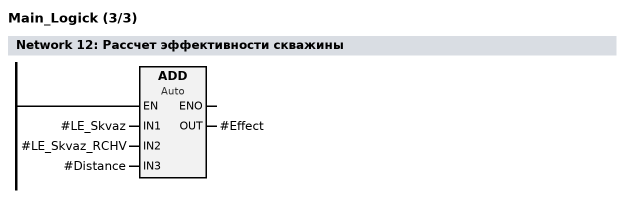
   RUNG wire#powerrail
      Add(in1 := #LE_Skvaz, in2 := #LE_Skvaz_RCHV, in3 := #Distance, out => #Effect)
   END_RUNG
   // the same network as SCL:
   #Effect := #LE_Skvaz + #LE_Skvaz_RCHV + #Distance;
END_REGION
END_FUNCTION_BLOCK

FUNCTION "Pump_LE" : Void
{ S7_Optimized_Access := 'TRUE' }
VERSION : 0.1
   VAR_INPUT 
      Level_Norm : Real;
      LS : Real;
      LE_now : Real;
   END_VAR

   VAR_TEMP 
      x : Array[1..10] of Real;
      Delta : Real;
   END_VAR


BEGIN
	//рассчёт коррекции при падении уровня в РЧВ
	#x[1] := #Level_Norm - #LS;
	#x[2] := #LE_now - #LS;
	#x[3] := #x[1] / #x[2];
	#Delta := 1 - #x[3];
	
	//уровень ниже рабочей точки
	IF #Delta < 1.0 THEN
	    "Main_Logick_DB".Alarms.LE_Warning := TRUE;
	ELSE
	    "Main_Logick_DB".Alarms.LE_Warning := FALSE;
	    #Delta := 1.0;
	END_IF;
	
	//уровень в аварийной зоне
	IF #Delta <= 0.0 THEN
	    "Main_Logick_DB".Alarms.LE_Alarm := TRUE;
	    #Delta := 0.0;
	ELSE
	    "Main_Logick_DB".Alarms.LE_Alarm := FALSE;
	END_IF;
	
	//коррекция уставки при аварийных ситуациях
	IF "Main_Logick_DB".Mode = TRUE THEN
	    "Pump_DB".SP_A := "Main_Logick_DB".PID_Pump.Result * #Delta;
	ELSE
	    "Pump_DB".SP_A := "Main_Logick_DB".SP_Pump * #Delta;
	END_IF;
END_FUNCTION

FUNCTION_BLOCK "DRV_Flow"   // FB130, LAD
{ S7_Optimized_Access := 'FALSE' }
VERSION : 0.1
// stored: AutoNumber false, IsIECCheckEnabled false, SetENOAutomatically false, UDAEnableTagReadback false
   VAR_IN_OUT
      impulse : Bool;
      FlowSpeed : Real;
   END_VAR
   VAR DB_SPECIFIC
      CMD : "CMD";
      Mode : Int;   // 0 - л/м, 1- л/ч, 2- м3/ч / Режим работы
      Status : Int;   // Статус устройства
      Use : Struct   // Функционал
         Indirect { S7_SetPoint := 'True'} : Bool := true;
         call_in_OB1 { S7_SetPoint := 'True'} : Bool := true;
      END_STRUCT;
      Clock { S7_SetPoint := 'True'} : Real := 0.1;   // Частота измерений
      Weight { S7_SetPoint := 'True'} : Real := 1.0;   // Вес импульса
      Time_Now : Real;
      Time_Last : Real;
      Time_Mid : Real;
      Flow_S : Real;   // литры в секунду
      Alarms : Word;   // Слово аварий
      Events : Word;   // События
      ADDR_BYTE { S7_SetPoint := 'True'} : Int;
      ADDR_BIT { S7_SetPoint := 'True'} : Int := 9;
   END_VAR
   VAR
      Filter { S7_SetPoint := 'True'} : "Filter";
   END_VAR
   VAR DB_SPECIFIC
      pos : Array[0..15] of Bool;
      "Name" { S7_SetPoint := 'True'} : String[4];
      Time_DTL : DTL;
   END_VAR
   VAR_TEMP
      imp : Bool;
      Filter_clock : Bool;
   END_VAR
   VAR CONSTANT
      sec : Int := 60;
   END_VAR
   // Filter.max := 100;
   VAR_TEMP   // added for the SCL form of the ladder/FBD networks
      _w1 : Bool;
      _w2 : Bool;
      _w3 : Bool;
   END_VAR
BEGIN

REGION Network 1: Чтение входа
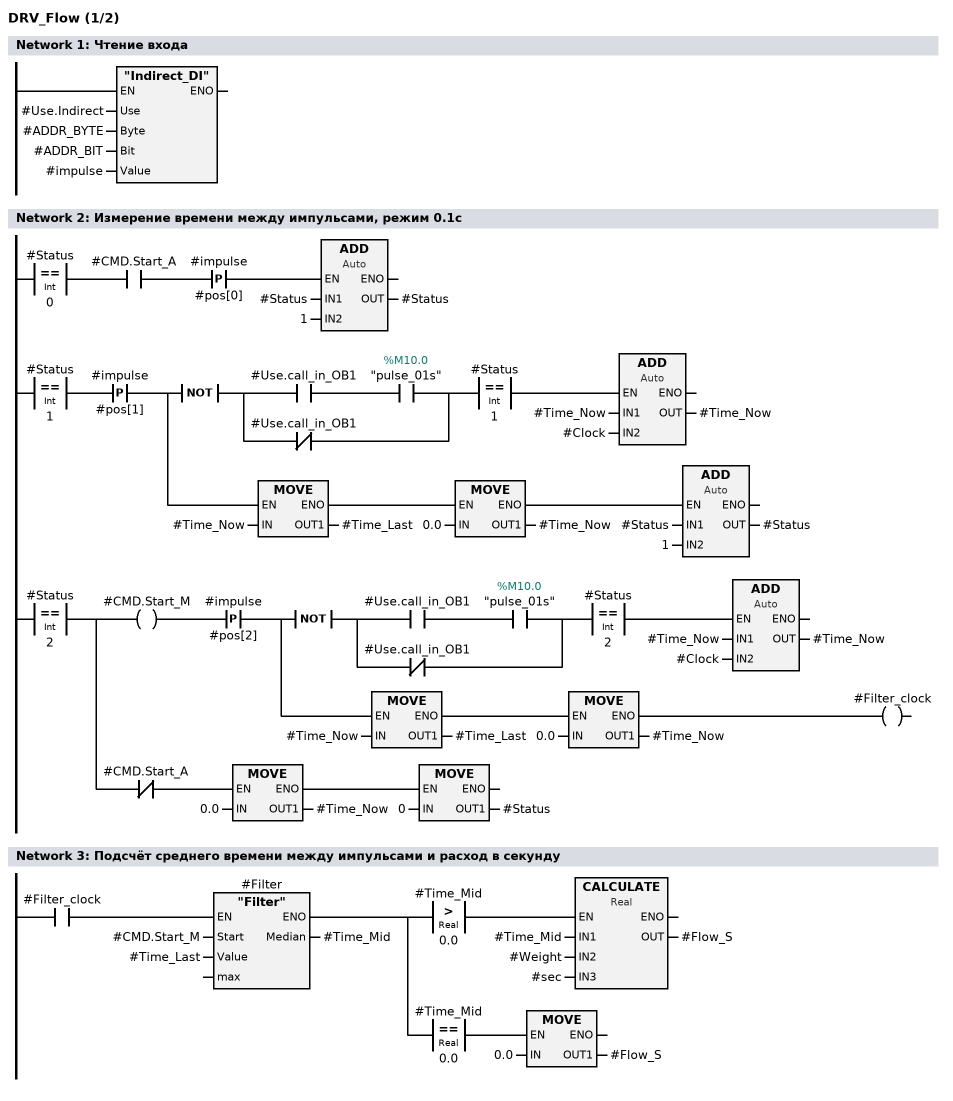
   RUNG wire#powerrail
      "Indirect_DI"(Use := #Use.Indirect, "Byte" := #ADDR_BYTE, Bit := #ADDR_BIT, Value := #impulse)
   END_RUNG
   // the same network as SCL:
   "Indirect_DI"(Use := #Use.Indirect, "Byte" := #ADDR_BYTE, Bit := #ADDR_BIT, Value := #impulse);
END_REGION

REGION Network 2: Измерение времени между импульсами, режим 0.1с
   RUNG wire#powerrail
      { S7_Templates := "SrcType := Int" } EQ_Contact(in1 := #Status, in2 := 0)
      Contact( #CMD.Start_A )
      P_Contact(operand := #impulse, bit := #pos[0])
      Add(in1 := #Status, in2 := 1, out => #Status)
   END_RUNG
   RUNG wire#powerrail
      { S7_Templates := "SrcType := Int" } EQ_Contact(in1 := #Status, in2 := 1)
      P_Contact(operand := #impulse, bit := #pos[1])
      wire#w1
      Not()
      wire#w2
      Contact( #Use.call_in_OB1 )
      Contact( "pulse_01s" )
      wire#w3
      { S7_Templates := "SrcType := Int" } EQ_Contact(in1 := #Status, in2 := 1)
      Add(in1 := #Time_Now, in2 := #Clock, out => #Time_Now)
   END_RUNG
   RUNG wire#w2
      I_Contact( #Use.call_in_OB1 )
   END_RUNG wire#w3
   RUNG wire#w1
      Move(in := #Time_Now, out1 => #Time_Last)
      Move(in := 0.0, out1 => #Time_Now)
      Add(in1 := #Status, in2 := 1, out => #Status)
   END_RUNG
   RUNG wire#powerrail
      { S7_Templates := "SrcType := Int" } EQ_Contact(in1 := #Status, in2 := 2)
      wire#w4
      Coil( #CMD.Start_M )
      P_Contact(operand := #impulse, bit := #pos[2])
      wire#w5
      Not()
      wire#w6
      Contact( #Use.call_in_OB1 )
      Contact( "pulse_01s" )
      wire#w7
      { S7_Templates := "SrcType := Int" } EQ_Contact(in1 := #Status, in2 := 2)
      Add(in1 := #Time_Now, in2 := #Clock, out => #Time_Now)
   END_RUNG
   RUNG wire#w6
      I_Contact( #Use.call_in_OB1 )
   END_RUNG wire#w7
   RUNG wire#w5
      Move(in := #Time_Now, out1 => #Time_Last)
      Move(in := 0.0, out1 => #Time_Now)
      Coil( #Filter_clock )
   END_RUNG
   RUNG wire#w4
      I_Contact( #CMD.Start_A )
      Move(in := 0.0, out1 => #Time_Now)
      Move(in := 0, out1 => #Status)
   END_RUNG
   // the same network as SCL:
   #_w1 := (#Status = 0) AND #CMD.Start_A AND #impulse AND NOT #pos[0];   // rising edge of #impulse
   #pos[0] := #impulse;
   IF #_w1 THEN #Status := #Status + 1; END_IF;
   #_w2 := (#Status = 1) AND #impulse AND NOT #pos[1];   // rising edge of #impulse
   #pos[1] := #impulse;
   IF NOT #_w2 AND ((#Use.call_in_OB1 AND "pulse_01s") OR NOT #Use.call_in_OB1) AND (#Status = 1) THEN
       #Time_Now := #Time_Now + #Clock;
   END_IF;
   IF #_w2 THEN
       #Time_Last := #Time_Now;
       #Time_Now := 0.0;
       #Status := #Status + 1;
   END_IF;
   #CMD.Start_M := #Status = 2;
   #_w3 := #CMD.Start_M AND #impulse AND NOT #pos[2];   // rising edge of #impulse
   #pos[2] := #impulse;
   IF NOT #_w3 AND ((#Use.call_in_OB1 AND "pulse_01s") OR NOT #Use.call_in_OB1) AND (#Status = 2) THEN
       #Time_Now := #Time_Now + #Clock;
   END_IF;
   IF #_w3 THEN
       #Time_Last := #Time_Now;
       #Time_Now := 0.0;
   END_IF;
   #Filter_clock := #_w3;
   IF #CMD.Start_M AND NOT #CMD.Start_A THEN
       #Time_Now := 0.0;
       #Status := 0;
   END_IF;
END_REGION

REGION Network 3: Подсчёт среднего времени между импульсами и расход в секунду
   RUNG wire#powerrail
      Contact( #Filter_clock )
      #Filter(Start := #CMD.Start_M, Value := #Time_Last, max :=, Median => #Time_Mid)
      wire#w1
      { S7_Templates := "SrcType := Real" } GT_Contact(in1 := #Time_Mid, in2 := 0.0)
      { S7_Templates := "SrcType := Real"; S7_Expression := "IN3/IN1*IN2" } Calculate(in1 := #Time_Mid, in2 := #Weight, in3 := #sec, out => #Flow_S)
   END_RUNG
   RUNG wire#w1
      { S7_Templates := "SrcType := Real" } EQ_Contact(in1 := #Time_Mid, in2 := 0.0)
      Move(in := 0.0, out1 => #Flow_S)
   END_RUNG
   // the same network as SCL:
   #Filter(EN := #Filter_clock, Start := #CMD.Start_M, Value := #Time_Last, Median => #Time_Mid, ENO => #_w1);   // "Filter"
   IF #_w1 AND (#Time_Mid > 0.0) THEN #Flow_S := #sec/#Time_Mid*#Weight; END_IF;
   IF #_w1 AND (#Time_Mid = 0.0) THEN #Flow_S := 0.0; END_IF;
END_REGION

REGION Network 4: Расход л/м, л/ч, м3/ч
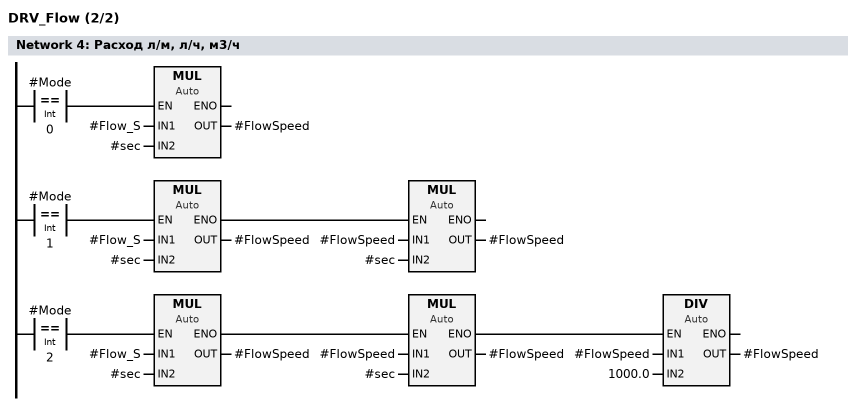
   RUNG wire#powerrail
      { S7_Templates := "SrcType := Int" } EQ_Contact(in1 := #Mode, in2 := 0)
      Mul(in1 := #Flow_S, in2 := #sec, out => #FlowSpeed)
   END_RUNG
   RUNG wire#powerrail
      { S7_Templates := "SrcType := Int" } EQ_Contact(in1 := #Mode, in2 := 1)
      Mul(in1 := #Flow_S, in2 := #sec, out => #FlowSpeed)
      Mul(in1 := #FlowSpeed, in2 := #sec, out => #FlowSpeed)
   END_RUNG
   RUNG wire#powerrail
      { S7_Templates := "SrcType := Int" } EQ_Contact(in1 := #Mode, in2 := 2)
      Mul(in1 := #Flow_S, in2 := #sec, out => #FlowSpeed)
      Mul(in1 := #FlowSpeed, in2 := #sec, out => #FlowSpeed)
      Div(in1 := #FlowSpeed, in2 := 1000.0, out => #FlowSpeed)
   END_RUNG
   // the same network as SCL:
   IF #Mode = 0 THEN #FlowSpeed := #Flow_S * #sec; END_IF;
   IF #Mode = 1 THEN
       #FlowSpeed := #Flow_S * #sec;
       #FlowSpeed := #FlowSpeed * #sec;
   END_IF;
   IF #Mode = 2 THEN
       #FlowSpeed := #Flow_S * #sec;
       #FlowSpeed := #FlowSpeed * #sec;
       #FlowSpeed := #FlowSpeed / 1000.0;
   END_IF;
END_REGION
END_FUNCTION_BLOCK

DATA_BLOCK "Comm_SKD1_DB"   // DB10
VERSION : 0.1
// stored: AutoNumber false, DBAccessibleFromOPCUA true, InstanceOfName Comm_SKD1, InstanceOfType FB
"Comm_SKD1"
BEGIN
   Valve_Name[1..10] := '';
END_DATA_BLOCK

DATA_BLOCK "Main_Logick_DB"   // DB1
VERSION : 0.1
// stored: AutoNumber true, DBAccessibleFromOPCUA true, InstanceOfName Main_Logick, InstanceOfType FB
"Main_Logick"
BEGIN
   PID_Pump.CMD.Vector := FALSE;
   PID_Pump.x := 1.0;
   PID_Pump.Settings.SP_P := 1.5;
   PID_Pump.Settings.SP_Ti := 150.0;
   PID_Pump.Settings.SP_Td := 0.0;
   PID_Pump.Settings.SP_Cycle := 0.2;
   PID_Pump.Settings.Max_SP := 500.0;
   PID_Pump.Settings.Min_SP := -500.0;
   PID_Pump.Settings.Max_in := 500.0;
   PID_Pump.Settings.Min_in := -500.0;
   PID_Pump.Settings.Max_out := 100.0;
   PID_Pump.Settings.Min_out := 0.0;
   PID_Pump.Settings.DeadBand := 1.0;
   PID_Pump.PID.IntegralResetMode := 4;
   PID_Pump.PID.RunModeByStartup := TRUE;
   PID_Pump.PID.SetSubstituteOutput := TRUE;
   PID_Pump.PID.ActivateRecoverMode := TRUE;
   PID_Pump.PID.CancelTuningLevel := 10.0;
   PID_Pump.PID.SubstituteOutput := 0.0;
   PID_Pump.PID.Config.InputPerOn := TRUE;
   PID_Pump.PID.Config.InvertControl := FALSE;
   PID_Pump.PID.Config.InputUpperLimit := 120.0;
   PID_Pump.PID.Config.InputLowerLimit := 0.0;
   PID_Pump.PID.Config.InputUpperWarning := 3.402822E+38;
   PID_Pump.PID.Config.InputLowerWarning := -3.402822E+38;
   PID_Pump.PID.Config.OutputUpperLimit := 100.0;
   PID_Pump.PID.Config.OutputLowerLimit := 0.0;
   PID_Pump.PID.Config.SetpointUpperLimit := 3.402822E+38;
   PID_Pump.PID.Config.SetpointLowerLimit := -3.402822E+38;
   PID_Pump.PID.Config.MinimumOnTime := 0.0;
   PID_Pump.PID.Config.MinimumOffTime := 0.0;
   PID_Pump.PID.Config.InputScaling.UpperPointIn := 27648.0;
   PID_Pump.PID.Config.InputScaling.LowerPointIn := 0.0;
   PID_Pump.PID.Config.InputScaling.UpperPointOut := 100.0;
   PID_Pump.PID.Config.InputScaling.LowerPointOut := 0.0;
   PID_Pump.PID.CycleTime.EnEstimation := TRUE;
   PID_Pump.PID.CycleTime.EnMonitoring := TRUE;
   PID_Pump.PID.CycleTime.Value := 0.1;
   PID_Pump.PID.CtrlParamsBackUp.Gain := 1.0;
   PID_Pump.PID.CtrlParamsBackUp.Ti := 20.0;
   PID_Pump.PID.CtrlParamsBackUp.Td := 0.0;
   PID_Pump.PID.CtrlParamsBackUp.TdFiltRatio := 0.2;
   PID_Pump.PID.CtrlParamsBackUp.PWeighting := 1.0;
   PID_Pump.PID.CtrlParamsBackUp.DWeighting := 1.0;
   PID_Pump.PID.CtrlParamsBackUp.Cycle := 1.0;
   PID_Pump.PID.PIDSelfTune.SUT.TuneRule := 0;
   PID_Pump.PID.PIDSelfTune.TIR.TuneRule := 0;
   PID_Pump.PID.Retain.CtrlParams.Gain := 1.0;
   PID_Pump.PID.Retain.CtrlParams.Ti := 20.0;
   PID_Pump.PID.Retain.CtrlParams.Td := 0.0;
   PID_Pump.PID.Retain.CtrlParams.TdFiltRatio := 0.2;
   PID_Pump.PID.Retain.CtrlParams.PWeighting := 1.0;
   PID_Pump.PID.Retain.CtrlParams.DWeighting := 1.0;
   PID_Pump.PID.Retain.CtrlParams.Cycle := 1.0;
   PID_Pump.C.SP := 1.0;
   PID_Pump.C.One := 0.1;
END_DATA_BLOCK

DATA_BLOCK "System_DB"   // DB4
VERSION : 0.1
// stored: AutoNumber true, DBAccessibleFromOPCUA true, InstanceOfName System, InstanceOfType FB
"System"
BEGIN
END_DATA_BLOCK

DATA_BLOCK "ModBus_DB"   // DB20
VERSION : 0.1
// stored: AutoNumber false, DBAccessibleFromOPCUA true, InstanceOfName ModBus, InstanceOfType FB
"ModBus"
BEGIN
END_DATA_BLOCK

DATA_BLOCK "ModBus_TCP_DB"   // DB40
VERSION : 0.1
// stored: AutoNumber false, DBAccessibleFromOPCUA true, InstanceOfName ModBus_TCP, InstanceOfType FB
"ModBus_TCP"
BEGIN
   DATA[0..100] := 16#0000;
   CONNECT.InterfaceId := 64;
   CONNECT.ID := 16#0001;
   CONNECT.ConnectionType := 16#0B;
   CONNECT.ActiveEstablished := TRUE;
   CONNECT.RemoteAddress.ADDR[1] := 16#0A;
   CONNECT.RemoteAddress.ADDR[2..3] := 16#01;
   CONNECT.RemoteAddress.ADDR[4] := 16#C9;
   CONNECT.RemotePort := 503;
   CONNECT.LocalPort := 0;
END_DATA_BLOCK

DATA_BLOCK "AIx_DB"   // DB220
VERSION : 0.1
// stored: AutoNumber false, DBAccessibleFromOPCUA true, InstanceOfName AIx, InstanceOfType FB
"AIx"
BEGIN
END_DATA_BLOCK

DATA_BLOCK "DIx_1_DB"   // DB200
VERSION : 0.1
// stored: AutoNumber false, DBAccessibleFromOPCUA true, InstanceOfName DIx_1, InstanceOfType FB
"DIx_1"
BEGIN
   AllBlock.Use.Inverse := FALSE;
   AllBlock.Use.Indirect := TRUE;
   AllBlock.ADDR_Byte := 0;
   AllBlock.ADDR_Bit := 3;
   AllBlock.Filter_On.SP := 16#02;
   AllBlock.Filter_Off.SP := 16#02;
   "3FOk".Use.Inverse := FALSE;
   "3FOk".Use.Indirect := TRUE;
   "3FOk".ADDR_Byte := 0;
   "3FOk".ADDR_Bit := 0;
   "3FOk".Filter_On.SP := 16#02;
   "3FOk".Filter_Off.SP := 16#02;
   Pump_Alarm.Use.Inverse := FALSE;
   Pump_Alarm.Use.Indirect := TRUE;
   Pump_Alarm.ADDR_Byte := 0;
   Pump_Alarm.ADDR_Bit := 2;
   Pump_Alarm.Filter_On.SP := 16#02;
   Pump_Alarm.Filter_Off.SP := 16#02;
   Leak_KP.Use.Inverse := FALSE;
   Leak_KP.Use.Indirect := TRUE;
   Leak_KP.ADDR_Byte := 0;
   Leak_KP.ADDR_Bit := 4;
   Leak_KP.Filter_On.SP := 16#02;
   Leak_KP.Filter_Off.SP := 16#02;
   Level_Norm.Use.Inverse := FALSE;
   Level_Norm.Use.Indirect := TRUE;
   Level_Norm.ADDR_Byte := 0;
   Level_Norm.ADDR_Bit := 5;
   Level_Norm.Filter_On.SP := 16#02;
   Level_Norm.Filter_Off.SP := 16#02;
   "3Fok_1".Use.Inverse := FALSE;
   "3Fok_1".Use.Indirect := TRUE;
   "3Fok_1".ADDR_Byte := 0;
   "3Fok_1".ADDR_Bit := 6;
   "3Fok_1".Filter_On.SP := 16#02;
   "3Fok_1".Filter_Off.SP := 16#02;
   "3Fok_2".Use.Inverse := FALSE;
   "3Fok_2".Use.Indirect := TRUE;
   "3Fok_2".ADDR_Byte := 0;
   "3Fok_2".ADDR_Bit := 7;
   "3Fok_2".Filter_On.SP := 16#02;
   "3Fok_2".Filter_Off.SP := 16#02;
   "3Fok_sh".Use.Inverse := FALSE;
   "3Fok_sh".Use.Indirect := TRUE;
   "3Fok_sh".ADDR_Byte := 1;
   "3Fok_sh".ADDR_Bit := 0;
   "3Fok_sh".Filter_On.SP := 16#02;
   "3Fok_sh".Filter_Off.SP := 16#02;
   SHUSKV_Ok.Use.Inverse := FALSE;
   SHUSKV_Ok.Use.Indirect := TRUE;
   SHUSKV_Ok.ADDR_Byte := 1;
   SHUSKV_Ok.ADDR_Bit := 1;
   SHUSKV_Ok.Filter_On.SP := 16#02;
   SHUSKV_Ok.Filter_Off.SP := 16#02;
   Leak_KP_res.Use.Inverse := FALSE;
   Leak_KP_res.Use.Indirect := TRUE;
   Leak_KP_res.ADDR_Byte := 1;
   Leak_KP_res.ADDR_Bit := 2;
   Leak_KP_res.Filter_On.SP := 16#02;
   Leak_KP_res.Filter_Off.SP := 16#02;
   Leak_KP_res_1.Use.Inverse := FALSE;
   Leak_KP_res_1.Use.Indirect := TRUE;
   Leak_KP_res_1.ADDR_Byte := 1;
   Leak_KP_res_1.ADDR_Bit := 3;
   Leak_KP_res_1.Filter_On.SP := 16#02;
   Leak_KP_res_1.Filter_Off.SP := 16#02;
   signal_12.Use.Inverse := FALSE;
   signal_12.Use.Indirect := TRUE;
   signal_12.ADDR_Byte := 0;
   signal_12.ADDR_Bit := 9;
   signal_12.Filter_On.SP := 16#02;
   signal_12.Filter_Off.SP := 16#02;
END_DATA_BLOCK

DATA_BLOCK "DOx_1_DB"   // DB210
VERSION : 0.1
// stored: AutoNumber false, DBAccessibleFromOPCUA true, InstanceOfName DOx_1, InstanceOfType FB
"DOx_1"
BEGIN
   All_Alarm.Use.Inverse := FALSE;
   All_Alarm.Use.Indirect := TRUE;
   All_Alarm.Use.Impulse := FALSE;
   All_Alarm.ADDR_Byte := 0;
   All_Alarm.ADDR_Bit := 1;
   All_Alarm.T_Impulse.SP := 16#02;
   command_2.Use.Inverse := FALSE;
   command_2.Use.Indirect := TRUE;
   command_2.Use.Impulse := FALSE;
   command_2.ADDR_Byte := 0;
   command_2.ADDR_Bit := 9;
   command_2.T_Impulse.SP := 16#02;
   command_3.Use.Inverse := FALSE;
   command_3.Use.Indirect := TRUE;
   command_3.Use.Impulse := FALSE;
   command_3.ADDR_Byte := 0;
   command_3.ADDR_Bit := 9;
   command_3.T_Impulse.SP := 16#02;
   command_4.Use.Inverse := FALSE;
   command_4.Use.Indirect := TRUE;
   command_4.Use.Impulse := FALSE;
   command_4.ADDR_Byte := 0;
   command_4.ADDR_Bit := 9;
   command_4.T_Impulse.SP := 16#02;
   command_5.Use.Inverse := FALSE;
   command_5.Use.Indirect := TRUE;
   command_5.Use.Impulse := FALSE;
   command_5.ADDR_Byte := 0;
   command_5.ADDR_Bit := 9;
   command_5.T_Impulse.SP := 16#02;
   command_6.Use.Inverse := FALSE;
   command_6.Use.Indirect := TRUE;
   command_6.Use.Impulse := FALSE;
   command_6.ADDR_Byte := 0;
   command_6.ADDR_Bit := 9;
   command_6.T_Impulse.SP := 16#02;
   command_7.Use.Inverse := FALSE;
   command_7.Use.Indirect := TRUE;
   command_7.Use.Impulse := FALSE;
   command_7.ADDR_Byte := 0;
   command_7.ADDR_Bit := 9;
   command_7.T_Impulse.SP := 16#02;
   command_8.Use.Inverse := FALSE;
   command_8.Use.Indirect := TRUE;
   command_8.Use.Impulse := FALSE;
   command_8.ADDR_Byte := 0;
   command_8.ADDR_Bit := 9;
   command_8.T_Impulse.SP := 16#02;
   command_9.Use.Inverse := FALSE;
   command_9.Use.Indirect := TRUE;
   command_9.Use.Impulse := FALSE;
   command_9.ADDR_Byte := 0;
   command_9.ADDR_Bit := 9;
   command_9.T_Impulse.SP := 16#02;
   command_10.Use.Inverse := FALSE;
   command_10.Use.Indirect := TRUE;
   command_10.Use.Impulse := FALSE;
   command_10.ADDR_Byte := 0;
   command_10.ADDR_Bit := 9;
   command_10.T_Impulse.SP := 16#02;
   command_11.Use.Inverse := FALSE;
   command_11.Use.Indirect := TRUE;
   command_11.Use.Impulse := FALSE;
   command_11.ADDR_Byte := 0;
   command_11.ADDR_Bit := 9;
   command_11.T_Impulse.SP := 16#02;
   command_12.Use.Inverse := FALSE;
   command_12.Use.Indirect := TRUE;
   command_12.Use.Impulse := FALSE;
   command_12.ADDR_Byte := 0;
   command_12.ADDR_Bit := 9;
   command_12.T_Impulse.SP := 16#02;
END_DATA_BLOCK

DATA_BLOCK "Motors_DB"   // DB240
VERSION : 0.1
// stored: AutoNumber false, DBAccessibleFromOPCUA true, InstanceOfName Motors, InstanceOfType FB
"Motors"
BEGIN
END_DATA_BLOCK

DATA_BLOCK "PID_Flow_DB"   // DB900
VERSION : 0.1
// stored: AutoNumber false, DBAccessibleFromOPCUA true, InstanceOfName PID_ex, InstanceOfType FB
"PID_ex"
BEGIN
   CMD.Vector := FALSE;
   PID.IntegralResetMode := 4;
   PID.RunModeByStartup := TRUE;
   PID.SetSubstituteOutput := TRUE;
   PID.ActivateRecoverMode := TRUE;
   PID.CancelTuningLevel := 10.0;
   PID.SubstituteOutput := 0.0;
   PID.Config.InputPerOn := FALSE;
   PID.Config.InvertControl := FALSE;
   PID.Config.InputUpperLimit := 500.0;
   PID.Config.InputLowerLimit := -500.0;
   PID.Config.InputUpperWarning := 3.402822E+38;
   PID.Config.InputLowerWarning := -3.402822E+38;
   PID.Config.OutputUpperLimit := 100.0;
   PID.Config.OutputLowerLimit := 0.0;
   PID.Config.SetpointUpperLimit := 500.0;
   PID.Config.SetpointLowerLimit := -500.0;
   PID.Config.MinimumOnTime := 0.0;
   PID.Config.MinimumOffTime := 0.0;
   PID.Config.InputScaling.UpperPointIn := 27648.0;
   PID.Config.InputScaling.LowerPointIn := 0.0;
   PID.Config.InputScaling.UpperPointOut := 100.0;
   PID.Config.InputScaling.LowerPointOut := 0.0;
   PID.CycleTime.EnEstimation := TRUE;
   PID.CycleTime.EnMonitoring := TRUE;
   PID.CycleTime.Value := 0.1;
   PID.CtrlParamsBackUp.Gain := 1.0;
   PID.CtrlParamsBackUp.Ti := 20.0;
   PID.CtrlParamsBackUp.Td := 0.0;
   PID.CtrlParamsBackUp.TdFiltRatio := 0.2;
   PID.CtrlParamsBackUp.PWeighting := 1.0;
   PID.CtrlParamsBackUp.DWeighting := 1.0;
   PID.CtrlParamsBackUp.Cycle := 1.0;
   PID.PIDSelfTune.SUT.TuneRule := 1;
   PID.PIDSelfTune.TIR.TuneRule := 0;
   PID.Retain.CtrlParams.Gain := 1.5;
   PID.Retain.CtrlParams.Ti := 150.0;
   PID.Retain.CtrlParams.Td := 0.0;
   PID.Retain.CtrlParams.TdFiltRatio := 0.2;
   PID.Retain.CtrlParams.PWeighting := 1.0;
   PID.Retain.CtrlParams.DWeighting := 1.0;
   PID.Retain.CtrlParams.Cycle := 1.0;
   C.SP := 0.2;
   C.One := 0.1;
END_DATA_BLOCK

DATA_BLOCK "PIDx_DB"   // DB260
VERSION : 0.1
// stored: AutoNumber false, DBAccessibleFromOPCUA true, InstanceOfName PIDx, InstanceOfType FB
"PIDx"
BEGIN
END_DATA_BLOCK

DATA_BLOCK "Pump_DB"   // DB600
VERSION : 0.1
// stored: AutoNumber false, DBAccessibleFromOPCUA true, InstanceOfName DRV_M_DA, InstanceOfType FB
"DRV_M_DA"
BEGIN
   Tx[0..1].SP := 0;
   Tx[2..3].SP := 10;
   Converter.Lim_High := FALSE;
   Converter.Lim_Low := FALSE;
   Converter.Inverse := FALSE;
   Converter.Min_In := 0.0;
   Converter.Min_Out := 0.0;
   Converter.Max_In := 50.0;
   Converter.Max_Out := 27648.0;
   Slow.Use_Up := FALSE;
   Slow.Use_Down := FALSE;
   Slow.Step_Up := 0.125;
   Slow.Step_Down := 0.125;
   Slow.T_Up.SP := 1.0;
   Slow.T_Up.One := 0.1;
   Slow.T_Down.SP := 1.0;
   Slow.T_Down.One := 0.1;
END_DATA_BLOCK

DATA_BLOCK "FB_DRV_Start_DB"   // DB100
VERSION : 0.1
// stored: AutoNumber false, DBAccessibleFromOPCUA true, InstanceOfName FB_DRV_Start, InstanceOfType FB
"FB_DRV_Start"
BEGIN
END_DATA_BLOCK

DATA_BLOCK "Time_SYS_DB"   // DB95
VERSION : 0.1
// stored: AutoNumber false, DBAccessibleFromOPCUA true, InstanceOfName Time_SYS, InstanceOfType FB
"Time_SYS"
BEGIN
   TimeZone.Bias := 180;
   TimeZone.DaylightBias := 60;
   TimeZone.DaylightStartMonth := 3;
   TimeZone.DaylightStartWeek := 5;
   TimeZone.DaylightStartWeekday := 7;
   TimeZone.DaylightStartHour := 2;
   TimeZone.DaylightStartMinute := 0;
   TimeZone.StandardStartMonth := 10;
   TimeZone.StandardStartWeek := 5;
   TimeZone.StandardStartWeekday := 1;
   TimeZone.StandardStartHour := 3;
   TimeZone.StandardStartMinute := 0;
   TimeZone.TimeZoneName := 'GMT+3';
   SET_TIMEZONE.REQ := FALSE;
   SET_TIMEZONE.TimeZone.Bias := 180;
   SET_TIMEZONE.TimeZone.DaylightBias := 60;
   SET_TIMEZONE.TimeZone.DaylightStartMonth := 3;
   SET_TIMEZONE.TimeZone.DaylightStartWeek := 5;
   SET_TIMEZONE.TimeZone.DaylightStartWeekday := 7;
   SET_TIMEZONE.TimeZone.DaylightStartHour := 2;
   SET_TIMEZONE.TimeZone.DaylightStartMinute := 0;
   SET_TIMEZONE.TimeZone.StandardStartMonth := 10;
   SET_TIMEZONE.TimeZone.StandardStartWeek := 5;
   SET_TIMEZONE.TimeZone.StandardStartWeekday := 1;
   SET_TIMEZONE.TimeZone.StandardStartHour := 3;
   SET_TIMEZONE.TimeZone.StandardStartMinute := 0;
   SET_TIMEZONE.TimeZone.TimeZoneName := 'GMT+3';
   SET_TIMEZONE.DONE := FALSE;
   SET_TIMEZONE.BUSY := FALSE;
   SET_TIMEZONE.ERROR := FALSE;
   SET_TIMEZONE.STATUS := 16#7000;
END_DATA_BLOCK

DATA_BLOCK "C_Pump_DB"   // DB300
VERSION : 0.1
// stored: AutoNumber false, DBAccessibleFromOPCUA true, InstanceOfName AI_ex, InstanceOfType FB
"AI_ex"
BEGIN
   Converter.Use_Min_In := FALSE;
   Converter.Use_Max_In := FALSE;
   Converter.Use_Min_Out := FALSE;
   Converter.Use_Max_Out := FALSE;
   Converter.IO := FALSE;
   Converter.Inverse := FALSE;
   Converter.Min_In := 0.0;
   Converter.Min_Out := 0.0;
   Converter.Max_In := 27648.0;
   Converter.Max_Out := 100.0;
   Tx[0..1].SP := 3.0;
   Tx[2..5].SP := 1.0;
   Tx[0..5].One := 0.1;
END_DATA_BLOCK

DATA_BLOCK "LE_DB"   // DB301
VERSION : 0.1
// stored: AutoNumber false, DBAccessibleFromOPCUA true, InstanceOfName AI_ex, InstanceOfType FB
"AI_ex"
BEGIN
   Converter.Use_Min_In := FALSE;
   Converter.Use_Max_In := FALSE;
   Converter.Use_Min_Out := FALSE;
   Converter.Use_Max_Out := FALSE;
   Converter.IO := FALSE;
   Converter.Inverse := FALSE;
   Converter.Min_In := 0.0;
   Converter.Min_Out := 0.0;
   Converter.Max_In := 27648.0;
   Converter.Max_Out := 100.0;
   Tx[0..1].SP := 3.0;
   Tx[2..5].SP := 1.0;
   Tx[0..5].One := 0.1;
END_DATA_BLOCK

DATA_BLOCK "PE_1_DB"   // DB304
VERSION : 0.1
// stored: AutoNumber false, DBAccessibleFromOPCUA true, InstanceOfName AI_ex, InstanceOfType FB
"AI_ex"
BEGIN
   Converter.Use_Min_In := FALSE;
   Converter.Use_Max_In := FALSE;
   Converter.Use_Min_Out := FALSE;
   Converter.Use_Max_Out := FALSE;
   Converter.IO := FALSE;
   Converter.Inverse := FALSE;
   Converter.Min_In := 0.0;
   Converter.Min_Out := 0.0;
   Converter.Max_In := 27648.0;
   Converter.Max_Out := 16.0;
   Tx[0..1].SP := 3.0;
   Tx[2..5].SP := 1.0;
   Tx[0..5].One := 0.1;
END_DATA_BLOCK

DATA_BLOCK "PE_2_DB"   // DB302
VERSION : 0.1
// stored: AutoNumber false, DBAccessibleFromOPCUA true, InstanceOfName AI_ex, InstanceOfType FB
"AI_ex"
BEGIN
   Converter.Use_Min_In := FALSE;
   Converter.Use_Max_In := FALSE;
   Converter.Use_Min_Out := FALSE;
   Converter.Use_Max_Out := FALSE;
   Converter.IO := FALSE;
   Converter.Inverse := FALSE;
   Converter.Min_In := 0.0;
   Converter.Min_Out := 0.0;
   Converter.Max_In := 27648.0;
   Converter.Max_Out := 16.0;
   Tx[0..1].SP := 3.0;
   Tx[2..5].SP := 1.0;
   Tx[0..5].One := 0.1;
END_DATA_BLOCK

DATA_BLOCK "PE_3_DB"   // DB303
VERSION : 0.1
// stored: AutoNumber false, DBAccessibleFromOPCUA true, InstanceOfName AI_ex, InstanceOfType FB
"AI_ex"
BEGIN
   Converter.Use_Min_In := FALSE;
   Converter.Use_Max_In := FALSE;
   Converter.Use_Min_Out := FALSE;
   Converter.Use_Max_Out := FALSE;
   Converter.IO := FALSE;
   Converter.Inverse := FALSE;
   Converter.Min_In := 0.0;
   Converter.Min_Out := 0.0;
   Converter.Max_In := 27648.0;
   Converter.Max_Out := 25.0;
   Tx[0..1].SP := 3.0;
   Tx[2..5].SP := 1.0;
   Tx[0..5].One := 0.1;
END_DATA_BLOCK

DATA_BLOCK "PE_4_DB"   // DB305
VERSION : 0.1
// stored: AutoNumber false, DBAccessibleFromOPCUA true, InstanceOfName AI_ex, InstanceOfType FB
"AI_ex"
BEGIN
   Converter.Use_Min_In := FALSE;
   Converter.Use_Max_In := FALSE;
   Converter.Use_Min_Out := FALSE;
   Converter.Use_Max_Out := FALSE;
   Converter.IO := FALSE;
   Converter.Inverse := FALSE;
   Converter.Min_In := 0.0;
   Converter.Min_Out := 0.0;
   Converter.Max_In := 27648.0;
   Converter.Max_Out := 25.0;
   Tx[0..1].SP := 3.0;
   Tx[2..5].SP := 1.0;
   Tx[0..5].One := 0.1;
END_DATA_BLOCK

DATA_BLOCK "TE_1_DB"   // DB306
VERSION : 0.1
// stored: AutoNumber false, DBAccessibleFromOPCUA true, InstanceOfName AI_ex, InstanceOfType FB
"AI_ex"
BEGIN
   Converter.Use_Min_In := FALSE;
   Converter.Use_Max_In := FALSE;
   Converter.Use_Min_Out := FALSE;
   Converter.Use_Max_Out := FALSE;
   Converter.IO := FALSE;
   Converter.Inverse := FALSE;
   Converter.Min_In := 0.0;
   Converter.Min_Out := -50.0;
   Converter.Max_In := 27648.0;
   Converter.Max_Out := 50.0;
   Tx[0..1].SP := 3.0;
   Tx[2..5].SP := 1.0;
   Tx[0..5].One := 0.1;
END_DATA_BLOCK

DATA_BLOCK "DB_Reset_All"   // DB1099
{ S7_Optimized_Access := 'TRUE' }
// stored: AutoNumber true, DBAccessibleFromOPCUA true, InstanceOfName IEC_TIMER, OfSystemLibElement IEC_TIMER, OfSystemLibVersion 1.0
"IEC_TIMER"
   // VAR
   //    PT : Time;
   //    ET { ExternalWritable := 'False'} : Time;
   //    IN : Bool;
   //    Q { ExternalWritable := 'False'} : Bool;
   // END_VAR
BEGIN
END_DATA_BLOCK

DATA_BLOCK "MB_CLIENT_DB"   // DB2
// stored: AutoNumber true, DBAccessibleFromOPCUA true, InstanceOfName MB_CLIENT, OfSystemLibElement MB_CLIENT, OfSystemLibVersion 5.2
"MB_CLIENT"
   // VAR_INPUT
   //    REQ : Bool;
   //    DISCONNECT : Bool;
   //    MB_MODE : USInt;
   //    MB_DATA_ADDR : UDInt;
   //    MB_DATA_LEN : UInt;
   // END_VAR
   // VAR_OUTPUT
   //    DONE : Bool;
   //    BUSY : Bool;
   //    ERROR : Bool;
   //    STATUS { ExternalVisible := 'False'} : Word;
   // END_VAR
   // VAR_IN_OUT
   //    MB_DATA_PTR : Variant;
   //    CONNECT : Variant;
   // END_VAR
   // VAR
   //    TCON { S7_SetPoint := 'True'} : TCON;
   //    TDISCON { S7_SetPoint := 'True'} : TDISCON;
   //    TSEND { S7_SetPoint := 'True'} : TSEND;
   //    TRECEIVE { S7_SetPoint := 'True'} : TRCV;
   //    TRESET { S7_SetPoint := 'True'} : T_RESET;
   //    TDIAG { S7_SetPoint := 'True'} : T_DIAG;
   //    TDIAG_Status { S7_SetPoint := 'True'} : TDiag_Status;
   //    Blocked_Proc_Timeout : Real;
   //    Rcv_Timeout : Real;
   //    MB_Unit_ID : Byte;
   //    MB_Transaction_ID : Word;
   //    MB_State { ExternalWritable := 'False'} : Word;
   //    SAVED_MB_DATA_ADDR : UDInt;
   //    SAVED_DATA_LEN : UInt;
   //    SAVED_MB_MODE : USInt;
   //    Connection_ID : Word;
   //    Retries : Word;
   //    TEMP_DATA { ExternalWritable := 'False'} : Array[1..263] of Byte;
   //    rcv_timer { ExternalAccessible := 'False'; ExternalVisible := 'False'; ExternalWritable := 'False'; S7_SetPoint := 'True'} : TON_TIME;
   //    wd_timer { ExternalAccessible := 'False'; ExternalVisible := 'False'; ExternalWritable := 'False'; S7_SetPoint := 'True'} : TON_TIME;
   //    Connected : Bool;
   //    Active { ExternalWritable := 'False'} : Bool;
   //    BytesReceived : UDInt;
   // END_VAR
BEGIN
END_DATA_BLOCK
